FUNCTION_BLOCK A24 EXTENDS GenericSubarea
VAR
	conveyors : ARRAY[1..6] OF POINTER TO Conveyor;
END_VAR
VAR
	step : (IDLE, RECEIVE, SEND, VACANT);
END_VAR

SUPER^();

CASE step OF
	IDLE:
		allConveyorsRequest(newRequest := ConveyorMode.IDLE);
		
		IF TRUE(*incoming bundle*) THEN
			step := RECEIVE;
		END_IF
		
	RECEIVE:
		allConveyorsRequest(newRequest := ConveyorMode.STOP);
		
		IF TRUE (*area 3 is done transferring*) THEN
			step := SEND;
		END_IF
		
	SEND:
		allConveyorsRequest(newRequest := ConveyorMode.FORWARD);
		
		IF allConveyorsVacant() THEN
			step := VACANT;
		END_IF
		
	VACANT:
		allConveyorsRequest(newRequest := ConveyorMode.IDLE);
		step := 0;
		
END_CASE

METHOD PROTECTED allConveyorsRequest : BOOL
VAR_INPUT
	newRequest : ConveyorMode;
END_VAR
VAR
	i : INT;
END_VAR
FOR i:=1 TO 6 BY 1 DO
	conveyors[i]^.setRequest(newRequest := newRequest);
END_FOR
END_METHOD

METHOD PROTECTED allConveyorsVacant : BOOL
VAR_INPUT
END_VAR
VAR
	i : INT;
END_VAR
FOR i:=1 TO 6 BY 1 DO
	IF conveyors[i]^.IsOccupied THEN
		RETURN;
	END_IF
END_FOR

allConveyorsVacant := TRUE;
END_METHOD

METHOD PROTECTED callHardware : BOOL
VAR_INPUT
END_VAR
END_METHOD

METHOD PROTECTED runModules : BOOL
VAR_INPUT
END_VAR
// NETWORK 1
END_METHOD

METHOD PROTECTED setupHardware : BOOL
VAR
	i : INT;
END_VAR
conveyors[1] := ADR(ConveyorSyncUnit.A24_LRC_C02);
conveyors[2] := ADR(ConveyorSyncUnit.A24_LRC_C04);
conveyors[3] := ADR(ConveyorSyncUnit.A24_LRC_C06);
conveyors[4] := ADR(ConveyorSyncUnit.A24_LRC_C08);
conveyors[5] := ADR(ConveyorSyncUnit.A24_LRC_C10);
conveyors[6] := ADR(ConveyorSyncUnit.A24_LRC_C12);
END_METHOD

END_FUNCTION_BLOCK

(* stored: Version 1.1.0.1, ProductVersion 3.1.4024.11
   POU A24: Id {9825abd9-77b4-48ca-9d54-54afdff6fff9}, SpecialFunc None
   Folder Conveyors: Id {8b2c3f28-68fb-4af7-bbe7-e360f5d9a9c4}
   Method allConveyorsRequest: Id {afc9e351-1478-4461-9636-ece7d59e3457}
   Method allConveyorsVacant: Id {11e98575-d900-40a7-b40a-04660dd3e276}
   Method callHardware: Id {c8ac936c-7d12-438b-a0a6-3c27a72b6d3c}
   Method runModules: Id {2010770a-d99d-45d5-a371-a2a4fae79adb}
   Method setupHardware: Id {4c5ab590-4716-4e6c-afb0-86b3c85cecc7} *)
